(* CODESYS project ccslib.library
   Company: ESO
   DocFormat: reStructuredText
   Description: ELT - CCS Library providing FB helping to receive deterministic data via MUDPI.
   Version: 0.0.0.6
   Placeholder: ESO ELT CCS Library
   Author: Mario Kiekebusch
   Title: ESO ELT CCS Library

Project tree, tasks and I/O mapping:
  libraries: ESO LDC Timer Library, * (ESO); ESO MUDPI Library, * (ESO); Tc2_EtherCAT, * (Beckhoff Automation GmbH); Tc2_Standard, * (Beckhoff Automation GmbH); Tc2_System, * (Beckhoff Automation GmbH); Tc2_Utilities, * (Beckhoff Automation GmbH); Tc3_Module, * (Beckhoff Automation GmbH); VisuDialogs, * (System); VisuSymbols, 3.5.10.0 (System)
  DUTs/
    Enumerated/
    Structures/
      data type T_CCS_GUI
      data type T_DATA_SAMPLE
      data type T_IP_ADDRESS
      data type T_PACKET_INFO
      data type T_TRACKING_DATA
      data type T_UDP_INFO
  GVLs/
    global variables GCL
    global variables GVL_TimeConstants
  lib/
  POUs/
    function F_Rad2Dms [ST]
    function F_Rad2Hms [ST]
    function block FB_CCS_RECEIVER [ST]: FB_init, GetParams, SetParams
    function block FB_LINEAR_INTERPOLATION [ST]: AddSample, Extrapolate, FB_init
    function block FB_MUDPI_RECEIVER [ST]: FB_exit, FB_init, FB_reinit, GetMudpiPayload, GetMudpiPayloadSize, GetTimestamp, IpAddressStringToInteger, IpIntegerToAddressString, ReceiveData, TcAddRef, TcQueryInterface, TcRelease, ValidatePacket
    function block FB_MUDPI_SENDER [ST]: FB_exit, FB_init, FB_reinit, ReceiveData, SendData, SetMudpiPayload, SetPacketInfo, SetTimestamp, TcAddRef, TcQueryInterface, TcRelease, UpdateMudpiPacket
    function IntegerToIpAddress [ST]
    function IpAdressToInteger [ST]
    program MAIN [ST]
  Version/
    global variables Global_Version
  VISUs/
    Templates/
      visualisation GUI_TEMPLATE_MUDPI_RECEIVER
      visualisation GUI_TEMPLATE_MUDPI_SENDER
  text list GlobalTextList
*)

// DUTs/Structures/T_CCS_GUI
TYPE T_CCS_GUI :
STRUCT
	alt: LREAL;
	az: LREAL;
	pa: LREAL;
	time_tai: STRING;
	lst: LREAL;
	ra: LREAL;
	dec: LREAL;
	nord_angle: LREAL;
	pupil_angle: LREAL;
	ha: LREAL;
END_STRUCT
END_TYPE

// DUTs/Structures/T_DATA_SAMPLE
TYPE T_DATA_SAMPLE :
STRUCT
	value: LREAL := 0.0;
	timestamp: LREAL := 0.0;
END_STRUCT
END_TYPE

// DUTs/Structures/T_IP_ADDRESS
TYPE T_IP_ADDRESS :
UNION
	ipAdrInternal : UDINT;
	ipAdr : ARRAY[0..3] OF BYTE;
END_UNION
END_TYPE

// DUTs/Structures/T_PACKET_INFO
TYPE T_PACKET_INFO :
STRUCT
	topicId: UDINT; 
	componentId: UINT; // counter the number of times the diagnostic data was sent.
	sampleId: UDINT; 
	frameId: UINT;
	numFrames: UINT;
	version: UINT;
	appTag: UINT;
	timestamp: LREAL;
	payloadSize: UINT;	
	size: UINT;
	valid: BOOL;
END_STRUCT
END_TYPE

// DUTs/Structures/T_TRACKING_DATA
TYPE T_TRACKING_DATA :
STRUCT
	
	target_observed_altaz : ARRAY [0..1] OF LREAL;
	current_observed_altaz : ARRAY [0..1] OF LREAL;
	time_lst : LREAL;
	time_tai : LREAL;
	time_utc : LREAL;
	north_angle : LREAL;
	pupil_angle : LREAL;
	elevation_direction_angle : LREAL;
	radec_at_altaz_at_requested_xy : ARRAY [0..1] OF LREAL;
	observed_altaz_at_requested_xy : ARRAY [0..1] OF LREAL;
	parallactic_angle : LREAL;
END_STRUCT
END_TYPE

// DUTs/Structures/T_UDP_INFO
TYPE T_UDP_INFO :
STRUCT
	bDriverInitialization: BOOL; // Indication of whether the realtime driver is properly initialized.  
	nReceivedPackets: UDINT; // counter the number of times the diagnostic data was sent.
	uSenderAddress: T_IP_ADDRESS;
	ipv4Adr : T_IPv4Addr := '';
	lrNotification: LREAL; // timestamp of the last sent
	sNotification: STRING;
END_STRUCT
END_TYPE

// GVLs/GCL
{attribute 'qualified_only'}
VAR_GLOBAL
	C_PI:				LREAL := 3.1415926535897932384626433832795028841971693993751;
    C_PI2: 				LREAL := C_PI / 2.0;
	C_2PI: 				LREAL := 2.0 * C_PI;
END_VAR

// GVLs/GVL_TimeConstants
{attribute 'qualified_only'}
VAR_GLOBAL
	C_INVALID:    DINT := -9999;
	C_ONE_SEC:    LINT := 1000000000;
	C_STAT_OK:    DINT := 0;
	C_NS2MSEC:    LREAL := 1/1E+6;
	C_NS2SEC:     LREAL := 1/1E+9;
	C_UNIX_OFFSET_SEC: ULINT := DATE_TO_ULINT(DATE#2000-01-01); // 946,684,800 seconds = 15,778,080 minutes = 262,968 hours
	C_UNIX_OFFSET_MICROSEC:  ULINT := C_UNIX_OFFSET_SEC * 10#1000_000;
END_VAR

// Version/Global_Version
{attribute 'TcGenerated'}
{attribute 'no-analysis'}
{attribute 'linkalways'}
// This function has been automatically generated from the project information.
VAR_GLOBAL CONSTANT
	{attribute 'const_non_replaced'}
	stLibVersion_ESO_ELT_CCS_Library : ST_LibVersion := (iMajor := 0, iMinor := 0, iBuild := 0, iRevision := 6, nFlags := 0, sVersion := '0.0.0.6');
END_VAR

// POUs/F_Rad2Dms
FUNCTION F_Rad2Dms : LREAL
VAR_INPUT
	dd:	LREAL;	// angle in radians
END_VAR
VAR
	value:		LREAL;
	degrees:	LINT;
	minutes:	LINT;
	seconds:	LREAL;
	dms: LREAL;
	
	sign:	int := 1;
END_VAR

IF dd < 0.0 THEN
	sign	:= -1;
	dd		:= -dd;
END_IF

value := dd / GCL.C_2PI * 360.0; 	// rad to degrees


degrees	:= TRUNC_INT(value);
minutes := TRUNC_INT((value - degrees)*60.0);
seconds := (value - degrees - minutes/60.0)*3600.0;

degrees	:= degrees * sign;	// put back the sign
dms := degrees * 10000.0 ;
dms := dms + (LINT_TO_LREAL(minutes) * 100.0 * sign);
dms := dms +  seconds * sign;
					
F_Rad2Dms	:= dms;

END_FUNCTION

// POUs/F_Rad2Hms
FUNCTION F_Rad2Hms : LREAL
VAR_INPUT
	hh:	LREAL;	// angle in radians
END_VAR
VAR
	value:		LREAL;
	hours:		INT;
	minutes:	INT;
	seconds:	LREAL;
	
	sign:	int := 1;
END_VAR

IF hh < 0.0 THEN
	sign	:= -1;
	hh		:= -hh;
END_IF

value := hh / GCL.C_2PI * 24.0; 	// rad to hours


hours	:= TRUNC_INT(value);
minutes := TRUNC_INT((value - hours)*60.0);
seconds := (value - hours - minutes/60.0)*3600.0;

hours	:= hours * sign;	// put back the sign

					
F_Rad2Hms	:= hours * 10000 + minutes * 100 + seconds;

END_FUNCTION

// POUs/FB_CCS_RECEIVER
FUNCTION_BLOCK FB_CCS_RECEIVER
VAR_INPUT
	refTimeObj  : REFERENCE TO FB_TIME; 
END_VAR
VAR_OUTPUT
END_VAR
VAR
	fbMudpiReceiver: FB_MUDPI_RECEIVER;
	tracking_raw : T_TRACKING_DATA;
	tracking_ccs : T_CCS_GUI;
	alt_sample: T_DATA_SAMPLE;
	pa_sample: T_DATA_SAMPLE;
	alt_angle_interpolator: FB_LINEAR_INTERPOLATION;
	pa_angle_interpolator: FB_LINEAR_INTERPOLATION;
	previous_sample_id: UDINT := 0;
	
	
  
	
	
END_VAR

fbMudpiReceiver();

// Get parameters
GetParams();

// Set parameters
SetParams();

METHOD FB_init : BOOL
VAR_INPUT
	bInitRetains : BOOL; // if TRUE, the retain variables are initialized (warm start / cold start)
	bInCopyCode : BOOL;  // if TRUE, the instance afterwards gets moved into the copy code (online change)
END_VAR
END_METHOD

METHOD GetParams
VAR_INPUT
END_VAR
VAR
	alt_angle_result : LREAL;
	pa_angle_result : LREAL;
	diff_time : LREAL;
END_VAR
IF (fbMudpiReceiver.packet_info.sampleId <> previous_sample_id) THEN
	memcpy(ADR(tracking_raw), fbMudpiReceiver.GetMudpiPayload(), fbMudpiReceiver.GetMudpiPayloadSize());
	alt_sample.value := tracking_raw.target_observed_altaz[0];
	alt_sample.timestamp := tracking_raw.time_tai;
	alt_angle_interpolator.AddSample(alt_sample);

	pa_sample.value := tracking_raw.parallactic_angle;
	pa_sample.timestamp := tracking_raw.time_tai;
	pa_angle_interpolator.AddSample(pa_sample);
	
	alt_angle_interpolator.Extrapolate(lrTimestamp:=refTimeObj.stat.lrTaiUnixTimeinSecs, lrValue=>alt_angle_result);
	pa_angle_interpolator.Extrapolate(lrTimestamp:=refTimeObj.stat.lrTaiUnixTimeinSecs, lrValue=>pa_angle_result);
	
	// Interpolating only PA and ALT for the time being. 
	// All the other tracking data are exactly as received.
	tracking_ccs.alt := RAD_TO_DEG(alt_angle_result);
	tracking_ccs.az := RAD_TO_DEG(tracking_raw.target_observed_altaz[1]);
	tracking_ccs.pa := RAD_TO_DEG(pa_angle_result);
	tracking_ccs.ra:= F_Rad2Hms(tracking_raw.radec_at_altaz_at_requested_xy[0]);
	tracking_ccs.dec := F_Rad2Dms(tracking_raw.radec_at_altaz_at_requested_xy[1]);
	tracking_ccs.pupil_angle := RAD_TO_DEG(tracking_raw.pupil_angle);
	tracking_ccs.nord_angle := RAD_TO_DEG(tracking_raw.north_angle);
	tracking_ccs.time_tai := DCTIME64_TO_STRING(refTimeObj.MudpiTimeToDc(tracking_raw.time_tai));
	tracking_ccs.ha := tracking_raw.time_lst - tracking_raw.radec_at_altaz_at_requested_xy[0];
	previous_sample_id := fbMudpiReceiver.packet_info.sampleId;
	diff_time := tracking_raw.time_tai - refTimeObj.stat.lrTaiUnixTimeinSecs;
ELSE
	alt_angle_interpolator.Extrapolate(lrTimestamp:=refTimeObj.stat.lrTaiUnixTimeinSecs, lrValue=>alt_angle_result);
	pa_angle_interpolator.Extrapolate(lrTimestamp:=refTimeObj.stat.lrTaiUnixTimeinSecs, lrValue=>pa_angle_result);
	
	alt_sample.value := alt_angle_result;
	alt_sample.timestamp := refTimeObj.stat.lrTaiUnixTimeinSecs;
	alt_angle_interpolator.AddSample(alt_sample);

	
	pa_sample.value := pa_angle_result;
	pa_sample.timestamp := refTimeObj.stat.lrTaiUnixTimeinSecs;
	pa_angle_interpolator.AddSample(pa_sample);
	
	tracking_ccs.alt := RAD_TO_DEG(alt_angle_result);
	tracking_ccs.pa := RAD_TO_DEG(pa_angle_result);
END_IF
END_METHOD

METHOD SetParams
VAR_INPUT
END_VAR
END_METHOD

END_FUNCTION_BLOCK

// POUs/FB_MUDPI_RECEIVER
(*
    This function blocks aims to CCS data coming in MUDPI frames.
    It uses the Beckhoff realtime UDP driver (TF6311). 
    The user of this function blocks needs to do the following in order for the library to work correctly:
    - Initialize the library with configuration parameters
        - Source port
*)

{attribute 'c++_compatible'}
FUNCTION_BLOCK FB_MUDPI_RECEIVER IMPLEMENTS ITcIoUdpProtocolRecv
VAR_INPUT
	port : UINT := 10000;
	instance_name: STRING := 'undefined';
END_VAR
VAR_OUTPUT
END_VAR
VAR
	(* TF6311 realtime driver parameters *)
    {attribute 'TcInitSymbol'}
    oid : OTCID;
    ipUdp : ITcIoUdpProtocol;
	nUdpPort : UINT := port;
    nReceivedPackets : UINT;
    uLastReceivedIP : T_IP_ADDRESS;
    hrInit : HRESULT;
    bSuccessfulInitializationOfRealtimeDriver : BOOL := FALSE; 
	(* Data/contents parameters *)
    mudpiPacket : ESO_MUDPI.FB_MudpiPacket(topicId := 300, componentId := 5);
	packet_info : T_PACKET_INFO;
	udp_info: T_UDP_INFO;
	sLibVersion:	   STRING	:= 'UNKNOWN'; // Library version
   

	
END_VAR

IF ipUdp <> 0 THEN
	ipUdp.CheckReceived();
END_IF

METHOD FB_exit : BOOL
VAR_INPUT
    bInCopyCode : BOOL; // if TRUE, the exit method is called for exiting an instance that is copied afterwards (online change).
END_VAR
IF NOT bInCopyCode THEN // no online change
    IF ipUdp <> 0 THEN
        //ipUdp.UnregisterReceiver(nUdpPort); // Shutdown
        ipUdp.UnregisterReceiver(nUdpPort); // Shutdown
        FW_SafeRelease(ADR(ipUdp));
        FB_exit := TRUE;
    END_IF
END_IF
END_METHOD

METHOD FB_init : BOOL
VAR_INPUT
    bInitRetains : BOOL; // if TRUE, the retain variables are initialized (warm start / cold start)
    bInCopyCode : BOOL;  // if TRUE, the instance afterwards gets moved into the copy code (online change)
END_VAR

sLibVersion := stLibVersion_ESO_ELT_CCS_Library.sVersion;

IF NOT bInCopyCode THEN // no online change
	IF ipUdp = 0 AND oid <> 0 THEN
	    hrInit := FW_ObjMgr_GetObjectInstance(	oid:=oid, 
											iid:=TC_GLOBAL_IID_LIST.IID_ITcIoUdpProtocol, 
											pipUnk:=ADR(ipUdp) );
		IF SUCCEEDED(hrInit) THEN 
			IF  SUCCEEDED(ipUdp.RegisterReceiver(nUdpPort, THIS^)) THEN //open port
				FB_init := TRUE;
				udp_info.bDriverInitialization := TRUE;
				(*bSuccessfulInitializationOfRealtimeDriver := TRUE;*)
			ELSE 
				FB_init := FALSE; 
				FW_SafeRelease(ADR(ipUdp));
			END_IF
		END_IF
	ELSIF oid = 0 THEN 
		FB_init := FALSE; 
		hrInit := ERR_INVALID_PARAM; 				
	END_IF
END_IF
END_METHOD

METHOD FB_reinit : BOOL
IF (ipUdp <> 0) THEN
    //ipUdp.RegisterReceiver(nUdpPort, THIS^);
    ipUdp.RegisterReceiver(nUdpPort, THIS^);
    FB_reinit := TRUE;
END_IF
END_METHOD

METHOD PUBLIC GetMudpiPayload : POINTER TO BYTE
GetMudpiPayload := mudpiPacket.GetPayload();
END_METHOD

METHOD PUBLIC GetMudpiPayloadSize : UINT
GetMudpiPayloadSize := mudpiPacket.GetPayloadSize();
END_METHOD

METHOD PUBLIC GetTimestamp : LREAL
VAR_INPUT	
END_VAR

GetTimestamp := packet_info.timestamp;
END_METHOD

METHOD PRIVATE IpAddressStringToInteger : UDINT
VAR_INPUT
    IpAddress : Tc2_System.T_IPv4Addr;
END_VAR
VAR
    IpAddressArray : Tc2_System.T_IPv4AddrArr;
    IpAddressInteger : UDINT;
END_VAR
IpAddressArray := Tc2_System.F_ScanIPv4AddrIds(sIPv4 := IpAddress);
IpAddressInteger := LREAL_TO_UDINT(IpAddressArray[0] * EXPT(256, 3) +
                                   IpAddressArray[1] * EXPT(256, 2) +
                                   IpAddressArray[2] * EXPT(256, 1) +
                                   IpAddressArray[3]);

IpAddressStringToInteger := IpAddressInteger;
END_METHOD

METHOD PRIVATE IpIntegerToAddressString : Tc2_System.T_IPv4Addr
VAR_INPUT
    IpAddress : T_IP_ADDRESS;
END_VAR
VAR
    IpAddressArray : Tc2_System.T_IPv4AddrArr;
	
END_VAR



IpAddressArray[3] := IpAddress.ipAdr[0];
IpAddressArray[2] := IpAddress.ipAdr[1];
IpAddressArray[1] := IpAddress.ipAdr[2];
IpAddressArray[0] := IpAddress.ipAdr[3];

IpIntegerToAddressString := F_CreateIPv4Addr( IpAddressArray );
END_METHOD

{attribute 'c++_compatible'}
{attribute 'minimal_input_size' := '4'}
{attribute 'pack_mode' := '4'}
{warning 'add method implementation'}
METHOD ReceiveData : HRESULT
VAR_INPUT
	ipAddr	: UDINT;
	udpDestPort	: UINT;
	udpSrcPort	: UINT;
	nData	: UDINT;
	pData	: PVOID;
	pVlan	: POINTER TO ETYPE_VLAN_HEADER := 0;
END_VAR
VAR
	tmp: LREAL;
END_VAR

VAR CONSTANT
	UNIX_OFFSET_MICROSEC: ULINT := DATE_TO_ULINT(DATE#2000-01-01) * 10#1000_000;
END_VAR
(*
nReceivedPackets := nReceivedPackets + 1;
uLastReceivedIP.ipAdrInternal := ipAddr;
memset(ADR(buffer), 0, SIZEOF(buffer));
memcpy(ADR(buffer), pData, nData);
*)
udp_info.nReceivedPackets := udp_info.nReceivedPackets + 1;
udp_info.uSenderAddress.ipAdrInternal := ipAddr;
udp_info.ipv4Adr := IpIntegerToAddressString(udp_info.uSenderAddress);

mudpiPacket.Initialize(inputData := pData,
                  size := UDINT_TO_UINT(nData));
packet_info.topicId := mudpiPacket.GetTopicId();
packet_info.componentId := mudpiPacket.GetComponentId();
packet_info.appTag := mudpiPacket.GetApplicationTag();
packet_info.version := mudpiPacket.GetVersion();
packet_info.frameId := mudpiPacket.GetFrameId();
packet_info.sampleId := mudpiPacket.GetSampleId();
packet_info.size := UDINT_TO_UINT(nData);
packet_info.payloadSize := mudpiPacket.GetPayloadSize();
packet_info.timestamp := mudpiPacket.GetTimestamp();
packet_info.valid := ValidatePacket();
END_METHOD

{attribute 'c++_compatible'}
{attribute 'minimal_input_size' := '4'}
{attribute 'pack_mode' := '4'}
{warning 'add method implementation'}
METHOD TcAddRef : UDINT
END_METHOD

{attribute 'object_name' := 'TcQueryInterface'}
{attribute 'c++_compatible'}
{attribute 'signature_flag' := '33554688'}
{attribute 'pack_mode' := '4'}
{attribute 'show'}
{attribute 'minimal_input_size' := '4'}
METHOD TcQueryInterface : HRESULT
VAR_INPUT
	iid	: REFERENCE TO IID;
	pipItf	: POINTER TO PVOID;
END_VAR
VAR
	ipUdpRecv : ITcIoUdpProtocolRecv;
	ipUnknown : ITcUnknown;	
END_VAR
IF GuidsEqual(ADR(iid), ADR(TC_GLOBAL_IID_LIST.IID_ITcIoUdpProtocolRecv)) THEN
	ipUdpRecv := THIS^; // cast to interface pointer
	pipItf^ := ITCUNKNOWN_TO_PVOID(ipUdpRecv);
	TcAddRef();
	TcQueryInterface := S_OK;
ELSIF GuidsEqual(ADR(iid), ADR(TC_GLOBAL_IID_LIST.IID_ITcUnknown)) THEN
	ipUnknown := THIS^; // cast to interface pointer
	pipItf^ := ITCUNKNOWN_TO_PVOID(ipUnknown);
	TcAddRef();
	TcQueryInterface := S_OK;
ELSE
	TcQueryInterface := E_HRESULTAdsErr.NOINTERFACE ; //Call super if this fb extends some other
END_IF
END_METHOD

{attribute 'c++_compatible'}
{attribute 'minimal_input_size' := '4'}
{attribute 'pack_mode' := '4'}
{warning 'add method implementation'}
METHOD TcRelease : UDINT
END_METHOD

(*
    This method verifies, if the checksum of a MUDPI packet is correct.
    TRUE = Checksum does match the content of the packet, FALSE = checksum does not match.
*)
METHOD PUBLIC ValidatePacket : BOOL
VAR
    checksum1 : UINT;
    checksum2 : UINT;
END_VAR

ValidatePacket := mudpiPacket.VerifyPacket();
END_METHOD

END_FUNCTION_BLOCK

// POUs/FB_LINEAR_INTERPOLATION
FUNCTION_BLOCK FB_LINEAR_INTERPOLATION
VAR_INPUT
END_VAR
VAR_OUTPUT
END_VAR
VAR
	x0:	T_DATA_SAMPLE;
	x1: T_DATA_SAMPLE;
	size:  UINT := 0;
END_VAR

METHOD AddSample : BOOL
VAR_INPUT
	sample: T_DATA_SAMPLE;
END_VAR

VAR
	
END_VAR
IF (size = 0) THEN
	x0 := sample;
	size := size + 1;
ELSIF (size = 1) THEN
	x1 := sample;
	size := size + 1;
ELSIF (size = 2) THEN
	x0 := x1;
	x1 := sample;
END_IF
END_METHOD

METHOD Extrapolate 
VAR_INPUT
lrTimestamp: LREAL;
END_VAR
VAR_OUTPUT
    bOk        : BOOL;
    lrValue    : LREAL;
END_VAR
VAR
	tmp        : LREAL;
END_VAR

tmp := x0.value + (lrTimestamp - x0.timestamp) / (x1.timestamp - x0.timestamp) * (x1.value - x0.value);
lrValue := tmp;
END_METHOD

METHOD FB_init : BOOL
VAR_INPUT
	bInitRetains : BOOL; // if TRUE, the retain variables are initialized (warm start / cold start)
	bInCopyCode : BOOL;  // if TRUE, the instance afterwards gets moved into the copy code (online change)
END_VAR
VAR
	sample: T_DATA_SAMPLE;
END_VAR
sample.value := 2.7;
sample.timestamp := 1.2;
AddSample(sample);
sample.value := 3.1;
sample.timestamp := 1.4;
AddSample(sample);
sample.value := 2.7;
sample.timestamp := 1.2;
AddSample(sample);
END_METHOD

END_FUNCTION_BLOCK

// POUs/FB_MUDPI_SENDER
(*
    This function blocks aims to pack the EL6688 diagnostic data in MUDPI frames
    and transmit them to Time System using Beckhoffs realtime UDP driver (TF6311). 
    The user of this function blocks needs to do the following in order for the library to work correctly:
    - Initialize the library with configuration parameters
        - Destination IP-address (a multicast address)
        - Destination port
        - Source port
*)

{attribute 'c++_compatible'}
FUNCTION_BLOCK FB_MUDPI_SENDER IMPLEMENTS ITcIoUdpProtocolRecv
VAR_INPUT
		ipAddress : Tc2_System.T_IPv4Addr := '0.0.0.0';
		dest_port : UINT := 10000;
		local_port : UINT := 20000;
		instance_name: STRING := 'undefined';
END_VAR
VAR_OUTPUT
END_VAR
VAR
	(* TF6311 realtime driver parameters *)
    {attribute 'TcInitSymbol'}
    oid : OTCID;
    ipUdp : ITcIoUdpProtocol;
    nReceivedPackets : UINT;
    uLastReceivedIP : T_IP_ADDRESS;
    hrInit : HRESULT;
    hrSend : HRESULT; 
    bSuccessfulInitializationOfRealtimeDriver : BOOL := FALSE; // Indication of whether the realtime driver is properly initialized.
	bEnableSending : BOOL := FALSE; // Indication of whether the sender is active or not.
	
	mudpiPacket : ESO_MUDPI.FB_MudpiPacket(topicId := 300, componentId := 5);
	packet_info : T_PACKET_INFO;
	
	  (* Transmission/communication parameters *)
	_destinationIpAddressString : Tc2_System.T_IPv4Addr;
    _destinationIpAddress : UDINT; // Destination address for the data
    _destinationPort : UINT; // Destination port for the data
    _sourcePort : UINT; // Source port of the data
	
	sLibVersion:	   STRING	:= 'UNKNOWN'; // Library version
	
END_VAR

(*
_destinationIpAddressString := ipAddress;
_destinationPort := dest_port;
_sourcePort := local_port;
*)

IF ipUdp <> 0 THEN
	ipUdp.CheckReceived();
END_IF

UpdateMudpiPacket();

METHOD FB_exit : BOOL
VAR_INPUT
    bInCopyCode : BOOL; // if TRUE, the exit method is called for exiting an instance that is copied afterwards (online change).
END_VAR
IF NOT bInCopyCode THEN // no online change
    IF ipUdp <> 0 THEN
        //ipUdp.UnregisterReceiver(nUdpPort); // Shutdown
        //ipUdp.UnregisterReceiver(nUdpPort); // Shutdown
        FW_SafeRelease(ADR(ipUdp));
        FB_exit := TRUE;
    END_IF
END_IF
END_METHOD

METHOD FB_init : BOOL
VAR_INPUT
    bInitRetains : BOOL; // if TRUE, the retain variables are initialized (warm start / cold start)
    bInCopyCode : BOOL;  // if TRUE, the instance afterwards gets moved into the copy code (online change)
END_VAR

sLibVersion := stLibVersion_ESO_ELT_CCS_Library.sVersion;
_destinationIpAddressString := ipAddress;
_destinationPort := dest_port;
_sourcePort := local_port;

IF NOT bInCopyCode THEN // no online change
	IF ipUdp = 0 AND oid <> 0 THEN
	    hrInit := FW_ObjMgr_GetObjectInstance(	oid:=oid, 
											iid:=TC_GLOBAL_IID_LIST.IID_ITcIoUdpProtocol, 
											pipUnk:=ADR(ipUdp) );
		
		IF SUCCEEDED(hrInit) THEN 
			bSuccessfulInitializationOfRealtimeDriver := TRUE;
		(*
			IF  SUCCEEDED(ipUdp.RegisterReceiver(nUdpPort, THIS^)) THEN //open port
				FB_init := TRUE;
			ELSE 
				FB_init := FALSE; 
				FW_SafeRelease(ADR(ipUdp));
			END_IF
			*)
		END_IF
		
	ELSIF oid = 0 THEN 
		FB_init := FALSE; 
		hrInit := ERR_INVALID_PARAM; 				
	END_IF
END_IF
END_METHOD

METHOD FB_reinit : BOOL
IF (ipUdp <> 0) THEN
    //ipUdp.RegisterReceiver(nUdpPort, THIS^);
    //ipUdp.RegisterReceiver(nUdpPort, THIS^);
    FB_reinit := TRUE;
END_IF
END_METHOD

{attribute 'c++_compatible'}
{attribute 'minimal_input_size' := '4'}
{attribute 'pack_mode' := '4'}
{warning 'add method implementation'}
METHOD ReceiveData : HRESULT
VAR_INPUT
	ipAddr	: UDINT;
	udpDestPort	: UINT;
	udpSrcPort	: UINT;
	nData	: UDINT;
	pData	: PVOID;
	pVlan	: POINTER TO ETYPE_VLAN_HEADER := 0;
END_VAR
nReceivedPackets := nReceivedPackets + 1;
uLastReceivedIP.ipAdrInternal := ipAddr;
END_METHOD

(*
    This method carry out the sending of the diagnostic data using the Ethernet network driver.
    The parameters are the array of data to be sent and the timestamp that is required by
	the MUDPI protocol.
*)

METHOD SendData : HRESULT
VAR_INPUT
END_VAR
	 
VAR
	
END_VAR

_DestinationIpAddress := IpAdressToInteger(_destinationIpAddressString);
IF ipUdp <> 0 AND bSuccessfulInitializationOfRealtimeDriver = TRUE AND bEnableSending THEN
						   
		// Send Data via UDP
    hrSend := ipUdp.SendData(ipDestAddr := _DestinationIpAddress,
                             udpDestPort := _DestinationPort,
                             udpSrcPort := _SourcePort,
                             nData := mudpiPacket.Size(),
                             pData := mudpiPacket.Data(),
                             bCalcUdpCheckSum := FALSE,
                             pVlan := 0);
    IF SUCCEEDED(hrSend) THEN
        mudpiPacket.IncreaseSampleId();
	END_IF
END_IF


SendData:= hrSend;
END_METHOD

METHOD PUBLIC SetMudpiPayload : BOOL
VAR_INPUT
    payload : POINTER TO BYTE;
    payloadSize : UINT;
END_VAR
SetMudpiPayload := mudpiPacket.SetPayload(payload, payloadSize);
END_METHOD

METHOD PUBLIC SetPacketInfo
VAR_INPUT
    TopicId : UDINT; // MUDPI Topic identity
    ComponentId : UINT; // MUDPI component identity
	Timestamp: LREAL := 0;
END_VAR
packet_info.topicId := TopicId;
packet_info.componentId := ComponentId;
packet_info.timestamp := Timestamp;
UpdateMudpiPacket();
END_METHOD

METHOD PUBLIC SetTimestamp
VAR_INPUT
	Timestamp: LREAL;
END_VAR
packet_info.timestamp := Timestamp;
mudpiPacket.SetTimestamp(packet_info.timestamp);
END_METHOD

{attribute 'c++_compatible'}
{attribute 'minimal_input_size' := '4'}
{attribute 'pack_mode' := '4'}
{warning 'add method implementation'}
METHOD TcAddRef : UDINT
END_METHOD

{attribute 'object_name' := 'TcQueryInterface'}
{attribute 'c++_compatible'}
{attribute 'signature_flag' := '33554688'}
{attribute 'pack_mode' := '4'}
{attribute 'show'}
{attribute 'minimal_input_size' := '4'}
METHOD TcQueryInterface : HRESULT
VAR_INPUT
	iid	: REFERENCE TO IID;
	pipItf	: POINTER TO PVOID;
END_VAR
VAR
	ipUdpRecv : ITcIoUdpProtocolRecv;
	ipUnknown : ITcUnknown;	
END_VAR
IF GuidsEqual(ADR(iid), ADR(TC_GLOBAL_IID_LIST.IID_ITcIoUdpProtocolRecv)) THEN
	ipUdpRecv := THIS^; // cast to interface pointer
	pipItf^ := ITCUNKNOWN_TO_PVOID(ipUdpRecv);
	TcAddRef();
	TcQueryInterface := S_OK;
ELSIF GuidsEqual(ADR(iid), ADR(TC_GLOBAL_IID_LIST.IID_ITcUnknown)) THEN
	ipUnknown := THIS^; // cast to interface pointer
	pipItf^ := ITCUNKNOWN_TO_PVOID(ipUnknown);
	TcAddRef();
	TcQueryInterface := S_OK;
ELSE
	TcQueryInterface := E_HRESULTAdsErr.NOINTERFACE ; //Call super if this fb extends some other
END_IF
END_METHOD

{attribute 'c++_compatible'}
{attribute 'minimal_input_size' := '4'}
{attribute 'pack_mode' := '4'}
{warning 'add method implementation'}
METHOD TcRelease : UDINT
END_METHOD

METHOD PUBLIC UpdateMudpiPacket
VAR_INPUT
END_VAR

mudpiPacket.SetTopicId(packet_info.topicId);
mudpiPacket.SetComponentId(packet_info.componentId);
mudpiPacket.SetTimestamp(packet_info.timestamp);
END_METHOD

END_FUNCTION_BLOCK

// POUs/IpAdressToInteger
FUNCTION IpAdressToInteger : UDINT
VAR_INPUT
	IpAddress : Tc2_System.T_IPv4Addr;
END_VAR
VAR
	IpAddressArray : Tc2_System.T_IPv4AddrArr;
    IpAddressInteger : UDINT;
END_VAR

IpAddressArray := Tc2_System.F_ScanIPv4AddrIds(sIPv4 := IpAddress);
IpAddressInteger := LREAL_TO_UDINT(IpAddressArray[0] * EXPT(256, 3) +
                                   IpAddressArray[1] * EXPT(256, 2) +
                                   IpAddressArray[2] * EXPT(256, 1) +
                                   IpAddressArray[3]);

IpAdressToInteger := IpAddressInteger;

END_FUNCTION

// POUs/IntegerToIpAddress
FUNCTION IntegerToIpAddress : Tc2_System.T_IPv4Addr
VAR_INPUT
	IpAddress : T_IP_ADDRESS;
END_VAR
VAR
	IpAddressArray : Tc2_System.T_IPv4AddrArr;
END_VAR


IpAddressArray[3] := IpAddress.ipAdr[0];
IpAddressArray[2] := IpAddress.ipAdr[1];
IpAddressArray[1] := IpAddress.ipAdr[2];
IpAddressArray[0] := IpAddress.ipAdr[3];

IntegerToIpAddress := F_CreateIPv4Addr( IpAddressArray );

END_FUNCTION

// POUs/MAIN
PROGRAM MAIN
VAR
	fbMudpiReceiver: FB_MUDPI_RECEIVER;
END_VAR

fbMudpiReceiver();

END_PROGRAM

// VISUs/Templates/GUI_TEMPLATE_MUDPI_RECEIVER
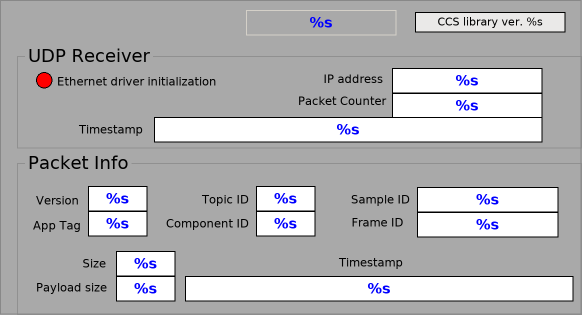
VISUALIZATION GUI_TEMPLATE_MUDPI_RECEIVER  // 582x315
VAR_INPUT
	m_DeviceName : STRING;
END_VAR
VAR_IN_OUT
	m_Instance : FB_MUDPI_RECEIVER;
END_VAR
    GroupBox (17,48 565x100), "UDP Receiver"
        Rectangle (375,20 150x25), "%s", text variable: m_Instance.udp_info.ipv4Adr
            OnMouseDown: write the text variable via Edit
        Label (285,18 84x26), "IP address"
        Label (37,19 240x29), "Ethernet driver initialization"
        Ellipse (19,24 16x16), tooltip "RED - False GREEN - True", colour toggle: m_Instance.udp_info.bDriverInitialization
        Label (265,40 107x26), "Packet Counter"
        Rectangle (375,45 150x25), "%s", text variable: m_Instance.udp_info.nReceivedPackets
            OnMouseDown: write the text variable via Edit
        Rectangle (137,69 388x25), "%s", tooltip "Time used for Simulation. Press "Copy UTC" or "Copy Local" button to get the time in correct format and then modify it for your needs.", text variable: m_Instance.udp_info.sNotification
            OnMouseDown: write the text variable via Default
        Label (56,70 76x23), "Timestamp"
    Rectangle (246,10 150x25), "%s", text variable: m_Instance.instance_name
    Rectangle (415,12 150x20), "CCS library ver. %s", text variable: m_Instance.sLibVersion
    GroupBox (17,155 565x160), "Packet Info"
        Rectangle (71,31 59x25), "%s", text variable: m_Instance.packet_info.version
            OnMouseDown: write the text variable via Edit
        Rectangle (71,56 59x25), "%s", text variable: m_Instance.packet_info.appTag
            OnMouseDown: write the text variable via Edit
        Label (6,31 59x29), "Version"
        Label (6,56 61x29), "App Tag"
        Label (329,30 67x29), "Sample ID"
        Rectangle (400,32 141x25), "%s", text variable: m_Instance.packet_info.sampleId
            OnMouseDown: write the text variable via Edit
        Rectangle (239,31 59x25), "%s", text variable: m_Instance.packet_info.topicId
            OnMouseDown: write the text variable via Edit
        Label (176,30 59x29), "Topic ID"
        Label (148,54 87x29), "Component ID"
        Rectangle (239,56 59x25), "%s", text variable: m_Instance.packet_info.componentId
            OnMouseDown: write the text variable via Edit
        Rectangle (400,57 141x25), "%s", text variable: m_Instance.packet_info.frameId
            OnMouseDown: write the text variable via Edit
        Label (304,53 89x29), "Frame ID"
        Label (316,96 76x23), "Timestamp"
        Rectangle (168,121 388x25), "%s", tooltip "Time used for Simulation. Press "Copy UTC" or "Copy Local" button to get the time in correct format and then modify it for your needs.", text variable: m_Instance.packet_info.timestamp
            OnMouseDown: write the text variable via Default
        Label (25,94 67x29), "Size"
        Label (12,118 81x29), "Payload size"
        Rectangle (99,96 59x25), "%s", text variable: m_Instance.packet_info.size
            OnMouseDown: write the text variable via Edit
        Rectangle (99,121 59x25), "%s", text variable: m_Instance.packet_info.payloadSize
            OnMouseDown: write the text variable via Edit
END_VISUALIZATION

// VISUs/Templates/GUI_TEMPLATE_MUDPI_SENDER
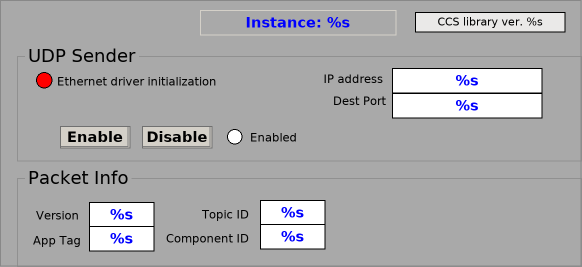
VISUALIZATION GUI_TEMPLATE_MUDPI_SENDER  // 582x267
VAR_INPUT
	m_DeviceName : STRING;
END_VAR
VAR_IN_OUT
	m_Instance : FB_MUDPI_SENDER;
END_VAR
    GroupBox (17,48 565x113), "UDP Sender"
        Rectangle (375,20 150x25), "%s", text variable: m_Instance._destinationIpAddressString
            OnMouseDown: write the text variable via Edit
        Label (285,18 84x26), "IP address"
        Label (37,19 240x29), "Ethernet driver initialization"
        Ellipse (19,24 16x16), tooltip "RED - False GREEN - True", colour toggle: m_Instance.bSuccessfulInitializationOfRealtimeDriver
        Label (265,40 107x26), "Dest Port"
        Rectangle (375,45 150x25), "%s", text variable: m_Instance._destinationPort
            OnMouseDown: write the text variable via Edit
        Button (43,78 70x22), "Enable", tooltip "Enable Diagnostics"
            OnMouseClick: execute { m_Instance.bEnableSending := TRUE; }
        Button (125,78 70x22), "Disable", tooltip "Disable Diagnostics"
            OnMouseClick: execute { m_Instance.bEnableSending := FALSE; }
        Label (230,75 61x29), "Enabled"
        Ellipse (210,81 15x15), tooltip "WHITE - Disabled GREEN - Enabled", colour toggle: m_Instance.bEnableSending
    Rectangle (200,10 196x25), "Instance: %s", text variable: m_Instance.instance_name
    Rectangle (415,12 150x20), "CCS library ver. %s", text variable: m_Instance.sLibVersion
    GroupBox (17,170 565x97), "Packet Info"
        Label (6,31 59x29), "Version"
        Label (6,56 61x29), "App Tag"
        Label (176,30 59x29), "Topic ID"
        Label (148,54 87x29), "Component ID"
        Rectangle (243,30 65x25), "%s", text variable: m_Instance.packet_info.topicId
            OnMouseDown: write the text variable via Edit
        Rectangle (243,54 65x25), "%s", text variable: m_Instance.packet_info.componentId
            OnMouseDown: write the text variable via Edit
        Rectangle (72,32 65x25), "%s", text variable: m_Instance.packet_info.version
            OnMouseDown: write the text variable via Edit
    Rectangle (89,226 65x25), "%s", text variable: m_Instance.packet_info.appTag
        OnMouseDown: write the text variable via Edit
END_VISUALIZATION
